(* IEC 61131-3 sources: programs/VI-54/VI-54_20171205/VI-54_20171205/Stations/PLC_VI54/VI-54_171014/Class/TestPositionTrigger, 1 file *)

(* ---- TestPositionTrigger.st ---- *)
(*!
<Class
	Name               = "TestPositionTrigger"
	Revision           = "1.1"
	RealtimeTask       = "false"
	CyclicTask         = "false"
	BackgroundTask     = "false"
	Sigmatek           = "false"
	OSInterface        = "false"
	HighPriority       = "false"
	Automatic          = "false"
	UpdateMode         = "Prescan"
	SharedCommandTable = "true"
	Objectsize         = "(480,240)">
	<Channels>
		<Server Name="ProdsPerMin" Visualized="true" Initialize="false" WriteProtected="false" Retentive="File"/>
		<Server Name="TestTriggerOn" Visualized="true" Initialize="false" WriteProtected="false" Retentive="false"/>
		<Server Name="Trigger" Visualized="true" Initialize="false" WriteProtected="true" Retentive="false"/>
		<Client Name="iActive" Required="false" Internal="false"/>
		<Client Name="iFcTrigger" Required="true" Internal="false"/>
		<Client Name="Position1" Required="false" Internal="false"/>
		<Client Name="Position2" Required="false" Internal="false"/>
		<Client Name="Position3" Required="false" Internal="false"/>
		<Client Name="Position4" Required="false" Internal="false"/>
		<Client Name="Position5" Required="false" Internal="false"/>
		<Client Name="STD" Required="true" Internal="true"/>
	</Channels>
	<Network Name="TestPositionTrigger">
		<!-- List of Components in this network -->
		<Components>
			<Object
				Name           = "STD"
				Class          = "Standard"
				Position       = "(210,360)"
				Visualized     = "false"
				BackgroundTime = "1000 ms">
				<Channels>
					<Server Name="ClassSvr"/>
				</Channels>
			</Object>
		</Components>
		<Comments>
		</Comments>
		<!-- List of Connections in this network -->
		<Connections>
			<Connection Source="this.STD" Destination="STD.ClassSvr"/>
		</Connections>
		<!-- Headerfiles -->
		<Options>
		</Options>
	</Network>
</Class>
*)
TestPositionTrigger : CLASS
  //Servers:
	Trigger 	: SvrChCmd_DINT;
	TestTriggerOn 	: SvrCh_DINT;
	ProdsPerMin 	: SvrCh_DINT;
  //Clients:
	iFcTrigger 	: CltCh_DINT;
	STD 	: CltChCmd_Standard;
	Position1 	: CltCh_DINT;
	Position2 	: CltCh_DINT;
	Position3 	: CltCh_DINT;
	Position4 	: CltCh_DINT;
	Position5 	: CltCh_DINT;
	iActive 	: CltCh_DINT;
  //Variables:
		Time_ms 	: UDINT;
		TmrMaintrigger 	: UDINT;
		NbrOfPositions 	: DINT;
		ActPosNbr 	: DINT;
  //Functions:

	FUNCTION GLOBAL PositionState
		VAR_OUTPUT
			State 	: ePosState;
		END_VAR;

	FUNCTION GLOBAL TestCycle
		VAR_OUTPUT
			State 	: TriggerStr;
		END_VAR;

	FUNCTION GLOBAL NormalCycle
		VAR_OUTPUT
			State 	: TriggerStr;
		END_VAR;

	FUNCTION GLOBAL ReadTrigger
		VAR_OUTPUT
			State 	: TriggerStr;
		END_VAR;

	FUNCTION GLOBAL SetNbrOfPositions
		VAR_INPUT
			Nbr 	: DINT;
		END_VAR;
  //Tables:
	FUNCTION @STD
		VAR_OUTPUT
			ret_code	: CONFSTATES;
		END_VAR;
	FUNCTION GLOBAL TAB @CT_;
END_CLASS;

#pragma using Standard

FUNCTION GLOBAL TestPositionTrigger::ReadTrigger
	VAR_OUTPUT
		State 	: TriggerStr;
	END_VAR

  // Is this funtion active?
  if IsClientConnected(#iActive) then
    iActive := iActive.Read();
  else
    iActive := 1;
  end_if;

  // Choose test cycle or normal cycle
  if iActive = 1 then
    if TestTriggerOn = 1 then
      State := TestCycle();
    else
      State := NormalCycle();
    end_if;
  end_if;

END_FUNCTION

FUNCTION GLOBAL TestPositionTrigger::PositionState
	VAR_OUTPUT
		State 	: ePosState;
	END_VAR

  if Position1.Read() = 1 then
    State := ePos1;
  elsif Position2.Read() = 1 then
    State := ePos2;
  elsif Position3.Read() = 1 then
    State := ePos3;
  elsif Position4.Read() = 1 then
    State := ePos4;
  elsif Position5.Read() = 1 then
    State := ePos5;
  end_if;

END_FUNCTION

FUNCTION GLOBAL TestPositionTrigger::TestCycle
	VAR_OUTPUT
		State 	: TriggerStr;
	END_VAR

  // Calculate timestamp
  if ProdsPerMin > 0 then
    Time_ms := 60000 / (to_udint ProdsPerMin);
  end_if;

  // Test cycle, choose position step by step
  if (ops.tAbsolute - TmrMaintrigger) >= Time_ms then
    if ActPosNbr >= NbrOfPositions then
      ActPosNbr := 0;
    end_if;
    ActPosNbr += 1;
    State.TriggerState  := 1;
    State.PositionState := ActPosNbr$ePosState;
    // Reset timer
    TmrMaintrigger := ops.tAbsolute;
  else
    State.TriggerState := 0;
  end_if;

  // Reset trigger state
//  if STD.TON(IN:= State.TriggerState, PT:= 20) then
//    State.TriggerState := 0;
//  end_if;

END_FUNCTION

FUNCTION GLOBAL TestPositionTrigger::NormalCycle
	VAR_OUTPUT
		State 	: TriggerStr;
	END_VAR

  State.PositionState := PositionState();
  State.TriggerState  := iFcTrigger.Read();

END_FUNCTION

FUNCTION GLOBAL TestPositionTrigger::SetNbrOfPositions
	VAR_INPUT
		Nbr 	: DINT;
	END_VAR

  NbrOfPositions := Nbr;

END_FUNCTION
